// TIA Portal project "Termico_Var_Erro" (V17)

(* hardware
DEVICE "S7-1200 station_1"  S7-1200 Station
   slot 0: "Rack_0"  S7-1200 Rack  Rack  V1.0
   slot 1: "PLC_1"  CPU 1214C AC/DC/Rly  6ES7 214-1BG40-0XB0  V4.0
   slot 3: "AQ 1x12BIT_1"  AQ1 signal board  6ES7 232-4HA30-0XB0  V1.0
*)

// ===== PLC "PLC_1"  CPU 1214C AC/DC/Rly =====

VAR_GLOBAL   // PLC tag table "Default tag table"
   "Sensor" AT %IW64 : Int;
   "Resultado" AT %MD10 : Real;
   "Temperatura_Atual" AT %MD14 : Real;
   "Temperatura_Anterior" AT %MD18 : Real;
   "Temperatura_Desejada" AT %MD22 : Real;
   "Erro_Temperatura" AT %MD26 : Real;
   "Variacao_do_Erro" AT %MD30 : Real;
   "PE_AN" AT %MD34 : Real;
   "PE_BN" AT %MD38 : Real;
   "PE_Z" AT %MD42 : Real;
   "PE_BP" AT %MD46 : Real;
   "PE_AP" AT %MD50 : Real;
   "PVE_NE" AT %MD54 : Real;
   "PVE_ZE" AT %MD58 : Real;
   "PVE_PO" AT %MD62 : Real;
   "Defuzzificada" AT %MD66 : Real;
   "Ventilador" AT %Q0.0 : Bool;
   "Saida_Analogica" AT %QW80 : Int;
   "Enable" AT %M100.0 : Bool;
   "Erro_Anterior" AT %MD70 : Real;
   "Resistencia" AT %MD74 : Real;
   "Resultado1" AT %MD78 : Real;
   "Ativa_Data_Log" AT %M200.0 : Bool;
   "Clock_Byte" AT %MB300 : Byte;
   "Clock_10Hz" AT %M300.0 : Bool;
   "Clock_5Hz" AT %M300.1 : Bool;
   "Clock_2.5Hz" AT %M300.2 : Bool;
   "Clock_2Hz" AT %M300.3 : Bool;
   "Clock_1.25Hz" AT %M300.4 : Bool;
   "Clock_1Hz" AT %M300.5 : Bool;
   "Clock_0.625Hz" AT %M300.6 : Bool;
   "Clock_0.5Hz" AT %M300.7 : Bool;
END_VAR

DATA_BLOCK "Data_block_1"   // DB3
{ S7_Optimized_Access := 'TRUE' }
VERSION : 0.1
   VAR
      records : UDInt := 30000;
      "name" : String := 'Dados';
      id : DWord := 1;
      header : String := 'Infos';
      data : Struct
         Temperatura_Atual : Real;
         Resistencia : Real;
         Temperatura_Desejada : Real;
         Erro_Temperatura : Real;
      END_STRUCT;
   END_VAR
   VAR RETAIN
      req : Bool;
   END_VAR
   VAR
      done : Bool;
      status : DWord;
   END_VAR
BEGIN
END_DATA_BLOCK

// folder: System blocks/Program resources

DATA_BLOCK "IEC_Timer_0_DB"   // DB1
{ S7_Optimized_Access := 'TRUE' }
AUTHOR : Simatic
FAMILY : IEC
NAME : IEC_TMR
VERSION : 1.0
// stored: InstanceOfName IEC_TIMER
"IEC_TIMER"
BEGIN
END_DATA_BLOCK

DATA_BLOCK "IEC_Timer_0_DB_1"   // DB2
{ S7_Optimized_Access := 'TRUE' }
AUTHOR : Simatic
FAMILY : IEC
NAME : IEC_TMR
VERSION : 1.0
// stored: InstanceOfName IEC_TIMER
"IEC_TIMER"
BEGIN
END_DATA_BLOCK

// folder: (top level)

FUNCTION "Fuzzifica" : Void   // FC1, SCL
{ S7_Optimized_Access := 'TRUE' }
VERSION : 0.1
   VAR_INPUT
      Erro_Temperatura : Real;
      Variacao_do_Erro : Real;
   END_VAR
   VAR_OUTPUT
      PE_AN : Real;
      PE_BN : Real;
      PE_ZE : Real;
      PE_BP : Real;
      PE_AP : Real;
      PVE_NE : Real;
      PVE_ZE : Real;
      PVE_PO : Real;
   END_VAR
BEGIN
   IF (#Erro_Temperatura >= -120) & (#Erro_Temperatura <= -40) THEN
       #PE_AN := 1;
       #PE_BN := 0;
       #PE_ZE := 0;
       #PE_BP := 0;
       #PE_AP := 0;
   END_IF;

   IF (#Erro_Temperatura >= -40) & (#Erro_Temperatura <= -20) THEN
       #PE_AN := ((-20 - #Erro_Temperatura) / 20);
       #PE_BN := ((#Erro_Temperatura + 40) / 20);
       #PE_ZE := 0;
       #PE_BP := 0;
       #PE_AP := 0;
   END_IF;

   IF (#Erro_Temperatura >= -20) & (#Erro_Temperatura <= 0) THEN
       #PE_AN := 0;
       #PE_BN := ((- #Erro_Temperatura) / 20);
       #PE_ZE := ((#Erro_Temperatura + 20) / 20);
       #PE_BP := 0;
       #PE_AP := 0;
   END_IF;

   IF (#Erro_Temperatura >= 0) & (#Erro_Temperatura <= 20) THEN
       #PE_AN := 0;
       #PE_BN := 0;
       #PE_ZE := ((20 - #Erro_Temperatura) / 20);
       #PE_BP := ((#Erro_Temperatura) / 20);
       #PE_AP := 0;
   END_IF;

   IF (#Erro_Temperatura >= 20) & (#Erro_Temperatura <= 40) THEN
       #PE_AN := 0;
       #PE_BN := 0;
       #PE_ZE := 0;
       #PE_BP := ((40 - #Erro_Temperatura) / 20);
       #PE_AP := ((#Erro_Temperatura - 20) / 20);
   END_IF;

   IF (#Erro_Temperatura >= 40) & (#Erro_Temperatura <= 120) THEN
       #PE_AN := 0;
       #PE_BN := 0;
       #PE_ZE := 0;
       #PE_BP := 0;
       #PE_AP := 1;
   END_IF;

   IF (#Variacao_do_Erro >= -30) & (#Variacao_do_Erro <= -5) THEN
       #PVE_NE := 1;
       #PVE_ZE := 0;
       #PVE_PO := 0;
   END_IF;

   IF (#Variacao_do_Erro >= -5) & (#Variacao_do_Erro <= 0) THEN
       #PVE_NE := (-1 * (#Variacao_do_Erro)) / 5;
       #PVE_ZE := (#Variacao_do_Erro + 5) / 5;
       #PVE_PO := 0;

   END_IF;

   IF (#Variacao_do_Erro >= 0) & (#Variacao_do_Erro <= 5) THEN
       #PVE_NE := 0;
       #PVE_ZE := (5 - #Variacao_do_Erro) / 5;
       #PVE_PO := (#Variacao_do_Erro) / 5;

   END_IF;

   IF (#Variacao_do_Erro >= 5) & (#Variacao_do_Erro <= 30) THEN
       #PVE_NE := 0;
       #PVE_ZE := 0;
       #PVE_PO := 1;

   END_IF;
END_FUNCTION

FUNCTION "Defuzzi" : Void   // FC2, SCL
{ S7_Optimized_Access := 'TRUE' }
VERSION : 0.1
   VAR_INPUT
      PE_AN : Real;
      PE_BN : Real;
      PE_Z : Real;
      PE_BP : Real;
      PE_AP : Real;
      PVE_NE : Real;
      PVE_ZE : Real;
      PVE_PO : Real;
   END_VAR
   VAR_OUTPUT
      Defuzzificada : Real;
   END_VAR
   VAR_TEMP
      Contador : Int;
      Vi : Real;
      Min1 : Real;
      Min2 : Real;
      Min3 : Real;
      Min4 : Real;
      Min5 : Real;
      Min6 : Real;
      Min7 : Real;
      Min8 : Real;
      Min9 : Real;
      Min10 : Real;
      Min11 : Real;
      Min12 : Real;
      Min13 : Real;
      Min14 : Real;
      Min15 : Real;
      Num : Real;
      Den : Real;
      V_MB : Array[0..500] of Real;
      V_B : Array[0..500] of Real;
      V_A : Array[0..500] of Real;
      V_MA : Array[0..500] of Real;
      V_X : Array[0..500] of Real;
      Agreg : Array[0..500] of Real;
      "#Contador := 0;#Vi := 0;WHILE #Contador <= 500 DO    #V_X[#Contador] := #Vi;    #Vi := #Vi + 0.02;    #Contador := #Contador + 1" : Array[0..500] of Real;
   END_VAR
BEGIN
   #Contador := 0;
   #Vi := 0;

   WHILE #Contador <= 500 DO
       #V_X[#Contador] := #Vi;
       #Vi := #Vi + 0.02;
       #Contador := #Contador + 1;
   END_WHILE;

   FOR #Contador := 0 TO 500 DO
       IF (#V_X[#Contador] >= 0) & (#V_X[#Contador] <= 1) THEN
           #V_MB[#Contador] := 1;
           #V_B[#Contador] := 0;
           #V_A[#Contador] := 0;
           #V_MA[#Contador] := 0;
       END_IF;

       IF (#V_X[#Contador] >= 1) & (#V_X[#Contador] <= 3) THEN
           #V_MB[#Contador] := (3 - #V_X[#Contador] / 2);
           #V_B[#Contador] := ((#V_X[#Contador] - 1) / 2);
           #V_A[#Contador] := 0;
           #V_MA[#Contador] := 0;
       END_IF;

       IF (#V_X[#Contador] >= 3) & (#V_X[#Contador] <= 5) THEN
           #V_MB[#Contador] := 0;
           #V_B[#Contador] := 1;
           #V_A[#Contador] := 0;
           #V_MA[#Contador] := 0;
       END_IF;

       IF (#V_X[#Contador] >= 5) & (#V_X[#Contador] <= 7) THEN
           #V_MB[#Contador] := 0;
           #V_B[#Contador] := ((7 - #V_X[#Contador]) / 2);
           ;
           #V_A[#Contador] := ((#V_X[#Contador]) - 5 / 2);
           #V_MA[#Contador] := 0;
       END_IF;

       IF (#V_X[#Contador] >= 7) & (#V_X[#Contador] <= 9) THEN
           #V_MB[#Contador] := 0;
           #V_B[#Contador] := 0;
           #V_A[#Contador] := ((9 - #V_X[#Contador]) / 2);
           #V_MA[#Contador] := ((#V_X[#Contador] - 7) / 2);
       END_IF;

       IF (#V_X[#Contador] >= 9) & (#V_X[#Contador] <= 10) THEN
           #V_MB[#Contador] := 0;
           #V_B[#Contador] := 0;
           #V_A[#Contador] := (10 - #V_X[#Contador]);
           #V_MA[#Contador] := 1;
       END_IF;

   END_FOR;


   #Min1 := MIN(IN1 := #PE_AN, IN2 := #PVE_NE);
   #Min2 := MIN(IN1 := #PE_BN, IN2 := #PVE_NE);
   #Min3 := MIN(IN1 := #PE_Z, IN2 := #PVE_NE);
   #Min4 := MIN(IN1 := #PE_BP, IN2 := #PVE_NE);
   #Min5 := MIN(IN1 := #PE_AP, IN2 := #PVE_NE);

   #Min6 := MIN(IN1 := #PE_AN, IN2 := #PVE_ZE);
   #Min7 := MIN(IN1 := #PE_BN, IN2 := #PVE_ZE);
   #Min8 := MIN(IN1 := #PE_Z, IN2 := #PVE_ZE);
   #Min9 := MIN(IN1 := #PE_BP, IN2 := #PVE_ZE);
   #Min10 := MIN(IN1 := #PE_AP, IN2 := #PVE_ZE);

   #Min11 := MIN(IN1 := #PE_AN, IN2 := #PVE_PO);
   #Min12 := MIN(IN1 := #PE_BN, IN2 := #PVE_PO);
   #Min13 := MIN(IN1 := #PE_Z, IN2 := #PVE_PO);
   #Min14 := MIN(IN1 := #PE_BP, IN2 := #PVE_PO);
   #Min15 := MIN(IN1 := #PE_AP, IN2 := #PVE_PO);


   //  Agregação da Regra 1,2
   FOR #Contador := 0 TO 500 DO
       #Agreg[#Contador] := MAX(IN1 := MIN(IN1 := #Min1, IN2 := #V_MB[#Contador]), IN2 := MIN(IN1 := #Min2, IN2 := #V_MB[#Contador]));
   END_FOR;

   //  Agregação da Regra 1,2 com a regra 3
   FOR #Contador := 0 TO 500 DO
       #Agreg[#Contador] := MAX(IN1 := #Agreg[#Contador], IN2 := MIN(IN1 := #Min3, IN2 := #V_MB[#Contador]));
   END_FOR;

   //  Agregação da Regra 1,2,3 com a regra 4
   FOR #Contador := 0 TO 500 DO
       #Agreg[#Contador] := MAX(IN1 := #Agreg[#Contador], IN2 := MIN(IN1 := #Min4, IN2 := #V_A[#Contador]));
   END_FOR;

   //  Agregação da Regra 1,2,3,4 com a regra 5
   FOR #Contador := 0 TO 500 DO
       #Agreg[#Contador] := MAX(IN1 := #Agreg[#Contador], IN2 := MIN(IN1 := #Min5, IN2 := #V_MA[#Contador]));
   END_FOR;

   //  Agregação da Regra 1,2,3,4,5 com a Regra 6
   FOR #Contador := 0 TO 500 DO
       #Agreg[#Contador] := MAX(IN1 := #Agreg[#Contador], IN2 := MIN(IN1 := #Min6, IN2 := #V_MB[#Contador]));
   END_FOR;

   //  Agregação da Regra 1,2,3,4,5,6 com a Regra 7
   FOR #Contador := 0 TO 500 DO
       #Agreg[#Contador] := MAX(IN1 := #Agreg[#Contador], IN2 := MIN(IN1 := #Min7, IN2 := #V_B[#Contador]));
   END_FOR;

   //  Agregação da Regra 1,2,3,4,5,6,7 com a Regra 8
   FOR #Contador := 0 TO 500 DO
       #Agreg[#Contador] := MAX(IN1 := #Agreg[#Contador], IN2 := MIN(IN1 := #Min8, IN2 := #V_MB[#Contador]));
   END_FOR;

   //  Agregação da Regra 1,2,3,4,5,6,7,8 com a Regra 9
   FOR #Contador := 0 TO 500 DO
       #Agreg[#Contador] := MAX(IN1 := #Agreg[#Contador], IN2 := MIN(IN1 := #Min9, IN2 := #V_A[#Contador]));
   END_FOR;

   //  Agregação da Regra 1,2,3,4,5,6,7,8,9 com a Regra 10
   FOR #Contador := 0 TO 500 DO
       #Agreg[#Contador] := MAX(IN1 := #Agreg[#Contador], IN2 := MIN(IN1 := #Min10, IN2 := #V_MA[#Contador]));
   END_FOR;

   //  Agregação da Regra 1,2,3,4,5,6,7,8,9,10 com a Regra 11
   FOR #Contador := 0 TO 500 DO
       #Agreg[#Contador] := MAX(IN1 := #Agreg[#Contador], IN2 := MIN(IN1 := #Min11, IN2 := #V_MB[#Contador]));
   END_FOR;

   //  Agregação da Regra 1,2,3,4,5,6,7,8,9,10,11 com a Regra 12
   FOR #Contador := 0 TO 500 DO
       #Agreg[#Contador] := MAX(IN1 := #Agreg[#Contador], IN2 := MIN(IN1 := #Min12, IN2 := #V_B[#Contador]));
   END_FOR;

   //  Agregação da Regra 1,2,3,4,5,6,7,8,9,10,11,12 com a Regra 13
   FOR #Contador := 0 TO 500 DO
       #Agreg[#Contador] := MAX(IN1 := #Agreg[#Contador], IN2 := MIN(IN1 := #Min13, IN2 := #V_MB[#Contador]));
   END_FOR;

   //  Agregação da Regra 1,2,3,4,5,6,7,8,9,10,11,12,13 com a Regra 14
   FOR #Contador := 0 TO 500 DO
       #Agreg[#Contador] := MAX(IN1 := #Agreg[#Contador], IN2 := MIN(IN1 := #Min14, IN2 := #V_A[#Contador]));
   END_FOR;

   //  Agregação da Regra 1,2,3,4,5,6,7,8,9,10,11,12,13,14 com a Regra 15
   FOR #Contador := 0 TO 500 DO
       #Agreg[#Contador] := MAX(IN1 := #Agreg[#Contador], IN2 := MIN(IN1 := #Min15, IN2 := #V_MA[#Contador]));
   END_FOR;

   // Esta sessão vai se destinar a realizar a defuzzificação pelo método da centróide (CoG), e assim determinar o valor de porcentagem de abertura da válvula de saída
   #Num := 0;
   #Den := 0;

   FOR #Contador := 0 TO 500 DO
       #Num := (#Num + (#Agreg[#Contador] * #V_X[#Contador]));
       #Den := (#Den + #Agreg[#Contador]);
   END_FOR;

   #Defuzzificada := (#Num) / (#Den);
END_FUNCTION

FUNCTION "Conversion" : Void   // FC3, SCL
{ S7_Optimized_Access := 'TRUE' }
VERSION : 0.1
   VAR_INPUT
      Erro_Temperatura : Real;
      Defuzzificada : Real;
   END_VAR
   VAR_OUTPUT
      Ventilador : Bool;
      Resistencia : Real;
   END_VAR
BEGIN
   IF (#Erro_Temperatura < 0) THEN
       #Resistencia := #Defuzzificada;
       #Ventilador := TRUE;
   END_IF;

   IF (#Erro_Temperatura>= 0) THEN
       #Resistencia := #Defuzzificada;
       #Ventilador := FALSE;
   END_IF;
END_FUNCTION

ORGANIZATION_BLOCK "Main"   // OB1, LAD, ProgramCycle
TITLE = "Main Program Sweep (Cycle)"
{ S7_Optimized_Access := 'TRUE' }
VERSION : 0.1
   VAR_INPUT
      Initial_Call : Bool;   // Initial call of this OB
      Remanence : Bool;   // =True, if remanent data are available
   END_VAR
   VAR_TEMP   // added for the SCL form of the ladder/FBD networks
      _w1 : Bool;
   END_VAR
BEGIN

REGION Network 1
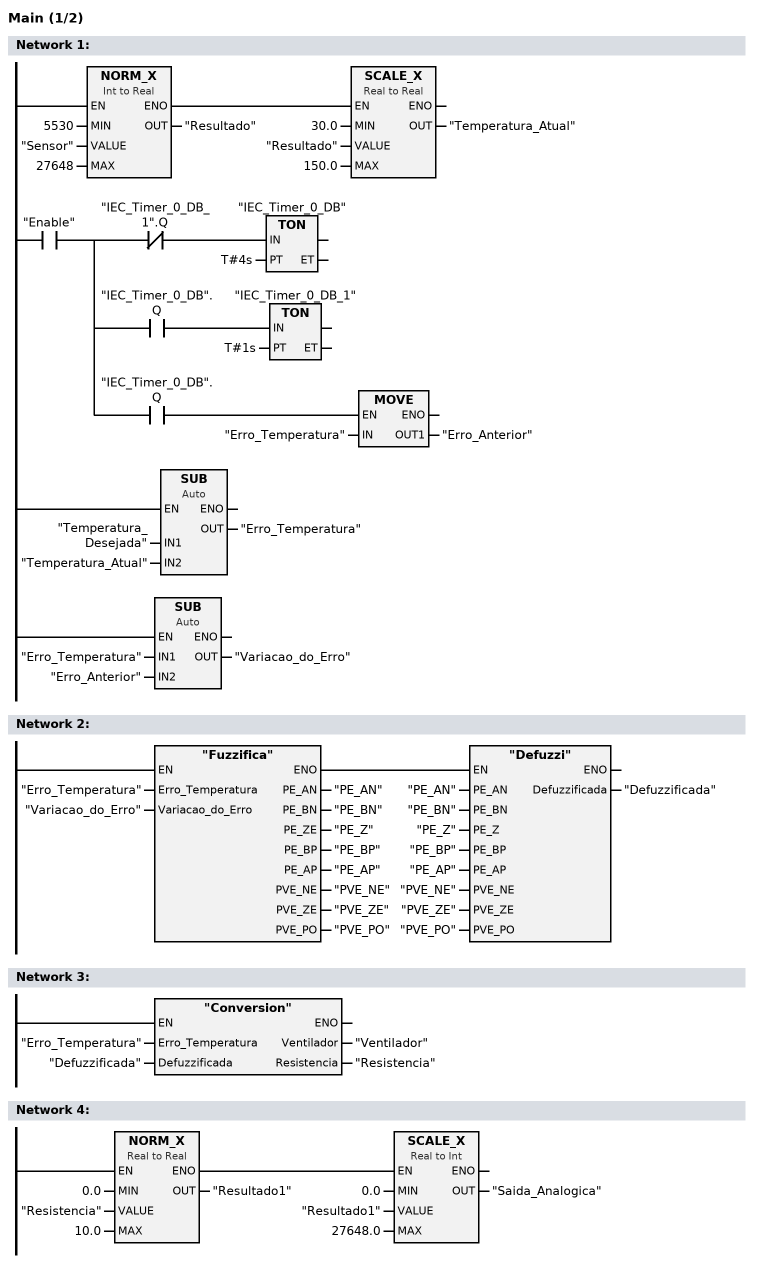
   "Resultado" := NORM_X(MIN := 5530, VALUE := "Sensor", MAX := 27648);
   "Temperatura_Atual" := SCALE_X(MIN := 30.0, VALUE := "Resultado", MAX := 150.0);
   "IEC_Timer_0_DB".TON(IN := "Enable" AND NOT "IEC_Timer_0_DB_1".Q, PT := T#4s);
   "IEC_Timer_0_DB_1".TON(IN := "Enable" AND "IEC_Timer_0_DB".Q, PT := T#1s);
   IF "Enable" AND "IEC_Timer_0_DB".Q THEN "Erro_Anterior" := "Erro_Temperatura"; END_IF;
   "Erro_Temperatura" := "Temperatura_Desejada" - "Temperatura_Atual";
   "Variacao_do_Erro" := "Erro_Temperatura" - "Erro_Anterior";
END_REGION

REGION Network 2
   RUNG wire#powerrail
      "Fuzzifica"(Erro_Temperatura := "Erro_Temperatura", Variacao_do_Erro := "Variacao_do_Erro", PE_AN => "PE_AN", PE_BN => "PE_BN", PE_ZE => "PE_Z", PE_BP => "PE_BP", PE_AP => "PE_AP", PVE_NE => "PVE_NE", PVE_ZE => "PVE_ZE", PVE_PO => "PVE_PO")
      "Defuzzi"(PE_AN := "PE_AN", PE_BN := "PE_BN", PE_Z := "PE_Z", PE_BP := "PE_BP", PE_AP := "PE_AP", PVE_NE := "PVE_NE", PVE_ZE := "PVE_ZE", PVE_PO := "PVE_PO", Defuzzificada => "Defuzzificada")
   END_RUNG
   // the same network as SCL:
   "Fuzzifica"(Erro_Temperatura := "Erro_Temperatura",
               Variacao_do_Erro := "Variacao_do_Erro",
               PE_AN => "PE_AN",
               PE_BN => "PE_BN",
               PE_ZE => "PE_Z",
               PE_BP => "PE_BP",
               PE_AP => "PE_AP",
               PVE_NE => "PVE_NE",
               PVE_ZE => "PVE_ZE",
               PVE_PO => "PVE_PO",
               ENO => #_w1);
   IF #_w1 THEN
       "Defuzzi"(PE_AN := "PE_AN",
                 PE_BN := "PE_BN",
                 PE_Z := "PE_Z",
                 PE_BP := "PE_BP",
                 PE_AP := "PE_AP",
                 PVE_NE := "PVE_NE",
                 PVE_ZE := "PVE_ZE",
                 PVE_PO := "PVE_PO",
                 Defuzzificada => "Defuzzificada");
   END_IF;
END_REGION

REGION Network 3
   RUNG wire#powerrail
      "Conversion"(Erro_Temperatura := "Erro_Temperatura", Defuzzificada := "Defuzzificada", Ventilador => "Ventilador", Resistencia => "Resistencia")
   END_RUNG
   // the same network as SCL:
   "Conversion"(Erro_Temperatura := "Erro_Temperatura",
                Defuzzificada := "Defuzzificada",
                Ventilador => "Ventilador",
                Resistencia => "Resistencia");
END_REGION

REGION Network 4
   RUNG wire#powerrail
      { S7_Templates := "[SrcType := Real, DestType := Real]" } Normalize(min := 0.0, value := "Resistencia", max := 10.0, out => "Resultado1")
      { S7_Templates := "[SrcType := Real, DestType := Int]" } Scale(min := 0.0, value := "Resultado1", max := 27648.0, out => "Saida_Analogica")
   END_RUNG
   // the same network as SCL:
   "Resultado1" := NORM_X(MIN := 0.0, VALUE := "Resistencia", MAX := 10.0);
   "Saida_Analogica" := SCALE_X(MIN := 0.0, VALUE := "Resultado1", MAX := 27648.0);
END_REGION

REGION Network 5
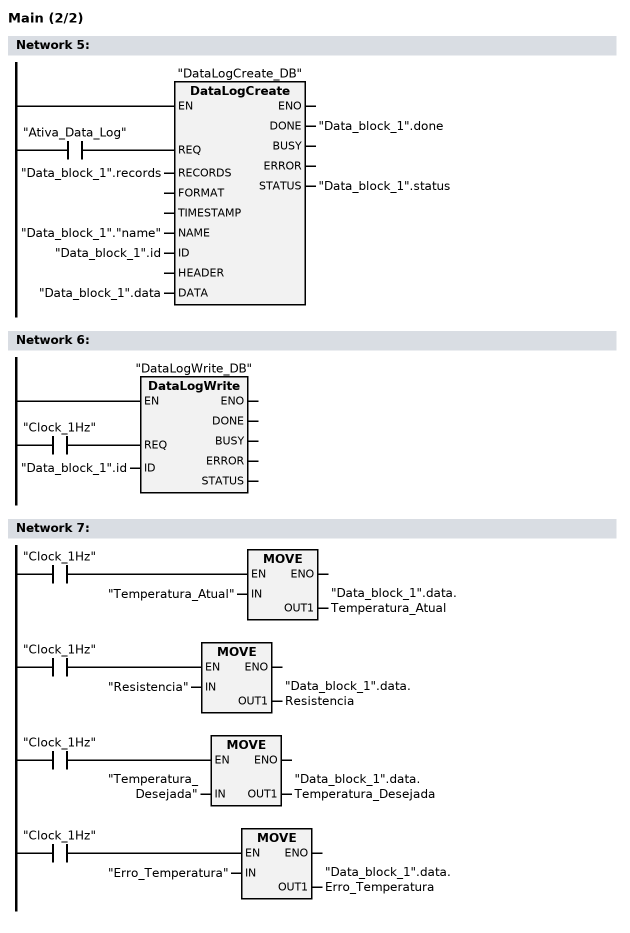
   "DataLogCreate_DB"(REQ := "Ativa_Data_Log",   // DataLogCreate
                      RECORDS := "Data_block_1".records,
                      "NAME" := "Data_block_1"."name",
                      ID := "Data_block_1".id,
                      DATA := "Data_block_1".data,
                      DONE => "Data_block_1".done,
                      STATUS => "Data_block_1".status);
END_REGION

REGION Network 6
   "DataLogWrite_DB"(REQ := "Clock_1Hz", ID := "Data_block_1".id);   // DataLogWrite
END_REGION

REGION Network 7
   RUNG wire#powerrail
      Contact( "Clock_1Hz" )
      Move(in := "Temperatura_Atual", out1 => "Data_block_1".data.Temperatura_Atual)
   END_RUNG
   RUNG wire#powerrail
      Contact( "Clock_1Hz" )
      Move(in := "Resistencia", out1 => "Data_block_1".data.Resistencia)
   END_RUNG
   RUNG wire#powerrail
      Contact( "Clock_1Hz" )
      Move(in := "Temperatura_Desejada", out1 => "Data_block_1".data.Temperatura_Desejada)
   END_RUNG
   RUNG wire#powerrail
      Contact( "Clock_1Hz" )
      Move(in := "Erro_Temperatura", out1 => "Data_block_1".data.Erro_Temperatura)
   END_RUNG
   // the same network as SCL:
   IF "Clock_1Hz" THEN
       "Data_block_1".data.Temperatura_Atual := "Temperatura_Atual";
       "Data_block_1".data.Resistencia := "Resistencia";
       "Data_block_1".data.Temperatura_Desejada := "Temperatura_Desejada";
       "Data_block_1".data.Erro_Temperatura := "Erro_Temperatura";
   END_IF;
END_REGION
END_ORGANIZATION_BLOCK